Staubli VAL3: new.pgx

public program new(string x_sName, num& x_nResult[])
  local string l_sPrefix
  local num l_nResult
begin
  // new one
end
